// TwinCAT 3 PLC project Untitled1
// ProgramVersion: 3.1.4023.0
// libraries:
//   Tc2_Standard, * (Beckhoff Automation GmbH)
//   Tc2_System, * (Beckhoff Automation GmbH)
//   Tc3_Module, * (Beckhoff Automation GmbH)
// project tree:
//   Abstract Factory/ FB_AbstractFactory.TcPOU (not stored)
//   / Class Diagram.TcCD (not stored), PlcTask.TcTTO
//   Colors/ FB_Black.TcPOU (not stored), FB_Red.TcPOU (not stored), FB_Yellow.TcPOU (not stored)
//   Creator/ FB_ColorCreator.TcPOU (not stored), FB_ShapeCreator.TcPOU, FB_ShapeCreatorEX.TcPOU (not stored)
//   DUTs/ E_Color.TcDUT (not stored), E_Factory.TcDUT, E_Shape.TcDUT (not stored)
//   Factory Producer/ FB_FactoryProducer.TcPOU
//   Interfaces/ I_Color.TcIO, I_Shape.TcIO (not stored)
//   POUs/ MAIN.TcPOU
//   Shapes/ FB_Circle.TcPOU (not stored), FB_CustomShape.TcPOU (not stored), FB_Rectangle.TcPOU, FB_Square.TcPOU (not stored), FB_Star.TcPOU (not stored), FB_Triangle.TcPOU (not stored)
// real-time tasks:
//   TASK PlcTask: cycle T#10ms, priority 20, ADS port 350

CONFIGURATION Untitled1
    RESOURCE PLC ON TwinCAT3
        TASK PlcTask(INTERVAL := T#10ms, PRIORITY := 20);
        PROGRAM MAIN WITH PlcTask : MAIN;
    END_RESOURCE
END_CONFIGURATION

// ---- DUTs/E_Factory.TcDUT
{attribute 'qualified_only'}
{attribute 'strict'}
TYPE E_Factory :
(
	init := 0,
	Shape,
	Color,
	end
);
END_TYPE

// ---- Interfaces/I_Color.TcIO
INTERFACE I_Color

METHOD M_Fill : BOOL
VAR_INPUT
END_VAR
END_METHOD

END_INTERFACE

// ---- POUs/MAIN.TcPOU
PROGRAM MAIN
VAR
	fbFactoryProducer : FB_FactoryProducer;
	fbFactory : REFERENCE TO FB_AbstractFactory;
	
	iShape : I_Shape;
	iColor : I_Color;
	
	eShape : E_Shape := E_Shape.Star;
	eColor : E_Color := E_Color.Red;
	
	bStart1: BOOL;	
	bStart2: BOOL;	
END_VAR

IF bStart1 THEN
	//Draw
	fbFactory REF= fbFactoryProducer.M_GetFactory(eFactory := E_Factory.Shape);
	
	IF __ISVALIDREF(fbFactory) THEN
		iShape := fbFactory.M_GetShapeObject(eShape:=eShape);
	END_IF
	
	IF iShape <> 0 THEN
		iShape.M_Draw();
	END_IF
	
	//Fill
	fbFactory REF= fbFactoryProducer.M_GetFactory(eFactory := E_Factory.Color);
	
	IF __ISVALIDREF(fbFactory) THEN
		iColor := fbFactory.M_GetColorObject(eColor:=eColor);
	END_IF
	
	IF iColor <> 0 THEN
		iColor.M_Fill();
	END_IF
	
	//Release Memory
	fbFactoryProducer.M_ReleaseMemory();
	
	bStart1 := FALSE;
END_IF

//Alternatively, you can chain the methods and get the same result: 
IF bStart2 THEN
	fbFactoryProducer.M_GetFactory(eFactory := E_Factory.Shape).M_GetShapeObject(eShape:=eShape).M_Draw();
	fbFactoryProducer.M_GetFactory(eFactory := E_Factory.Color).M_GetColorObject(eColor:=eColor).M_Fill();
	
	//Release Memory
	fbFactoryProducer.M_ReleaseMemory();
	bStart2 := FALSE;
END_IF

END_PROGRAM

// ---- Factory Producer/FB_FactoryProducer.TcPOU
FUNCTION_BLOCK FB_FactoryProducer
VAR_INPUT
END_VAR
VAR_OUTPUT
END_VAR
VAR
	pColorFactoy : POINTER TO FB_ColorCreator;
	pShapeFactory : POINTER TO FB_ShapeCreator;
END_VAR

METHOD FB_exit : BOOL
VAR_INPUT
	bInCopyCode : BOOL; // if TRUE, the exit method is called for exiting an instance that is copied afterwards (online change).
END_VAR
IF pColorFactoy <> 0 THEN
	__DELETE(pColorFactoy);
	pColorFactoy := 0;
END_IF

IF pShapeFactory <> 0 THEN
	__DELETE(pShapeFactory);
	pShapeFactory := 0;
END_IF
END_METHOD

METHOD M_GetFactory : REFERENCE TO FB_AbstractFactory
VAR_INPUT
	eFactory : E_Factory;
END_VAR
CASE eFactory OF
	E_Factory.Color:
	
		pColorFactoy := __NEW(FB_ColorCreator);
		IF pColorFactoy <> 0 THEN
			M_GetFactory REF= (pColorFactoy^);
		END_IF
	
		eFactory := E_Factory.init;
	
	E_Factory.Shape:
	
		pShapeFactory := __NEW(FB_ShapeCreator);
		IF pShapeFactory <> 0 THEN
			M_GetFactory REF= (pShapeFactory^);
		END_IF

		eFactory := E_Factory.init;
	
END_CASE
END_METHOD

METHOD M_ReleaseMemory : BOOL
VAR_INPUT
END_VAR
IF pColorFactoy <> 0 THEN
	__DELETE(pColorFactoy);
	pColorFactoy := 0;
END_IF

IF pShapeFactory <> 0 THEN
	__DELETE(pShapeFactory);
	pShapeFactory := 0;
END_IF
END_METHOD

END_FUNCTION_BLOCK

// ---- Creator/FB_ShapeCreator.TcPOU
{attribute 'hide_all_locals'}
{attribute 'enable_dynamic_creation'}
FUNCTION_BLOCK FB_ShapeCreator  EXTENDS FB_AbstractFactory
VAR_INPUT
END_VAR
VAR_OUTPUT
END_VAR
VAR
      pCircle    : POINTER TO FB_Circle;
      pRectangle : POINTER TO FB_Rectangle;
      pSquare    : POINTER TO FB_Square;
      pStar      : POINTER TO FB_Star;
      pTriangle  : POINTER TO FB_Triangle;
      iShape 	 : I_Shape;
END_VAR

METHOD FB_exit : BOOL
VAR_INPUT
	bInCopyCode : BOOL; // if TRUE, the exit method is called for exiting an instance that is copied afterwards (online change).
END_VAR
IF (pCircle <> 0) THEN
  __DELETE(pCircle);
  pCircle := 0;
END_IF

IF (pRectangle <> 0) THEN
  __DELETE(pRectangle);
  pRectangle := 0;
END_IF

IF (pSquare <> 0) THEN
  __DELETE(pSquare);
  pSquare := 0;
END_IF

IF (pStar <> 0) THEN
  __DELETE(pStar);
  pStar := 0;
END_IF

IF (pTriangle <> 0) THEN
  __DELETE(pTriangle);
  pTriangle := 0;
END_IF
END_METHOD

METHOD M_GetShapeObject : I_shape
VAR_INPUT
	eShape : E_Shape;
END_VAR
CASE eShape OF
	E_Shape.Circle:
		
		//Dynamic instantiation  
		pCircle := __NEW(FB_Circle);
		iShape := pCircle^;
		
		//Return the object
		IF iShape <> 0 THEN
			M_GetShapeObject := iShape;
		END_IF
		
		//Release the memory
		IF (pCircle <> 0) THEN
			__DELETE(pCircle);
			pCircle := 0;
		END_IF
		
		eShape := E_Shape.init;
	
	E_Shape.Rectangle:
		pRectangle := __NEW(FB_Rectangle);
		iShape := pRectangle^;
		
		//Return the object
		IF iShape <> 0 THEN
			M_GetShapeObject := iShape;
		END_IF
		
		IF (pRectangle <> 0) THEN
			__DELETE(pRectangle);
			pRectangle := 0;
		END_IF
		
		eShape := E_Shape.init;	
		
	E_Shape.Sqaure:
		pSquare := __NEW(FB_Square);
		iShape := pSquare^;
		
		//Return the object
		IF iShape <> 0 THEN
			M_GetShapeObject := iShape;
		END_IF
		
		IF (pSquare <> 0) THEN
			__DELETE(pSquare);
			pSquare := 0;
		END_IF
		
		eShape := E_Shape.init;	

	E_Shape.Star:
		pStar := __NEW(FB_Star);
		iShape := pStar^;
		
		//Return the object
		IF iShape <> 0 THEN
			M_GetShapeObject := iShape;
		END_IF
		
		IF (pStar <> 0) THEN
			__DELETE(pStar);
			pStar := 0;
		END_IF
		
		eShape := E_Shape.init;	
	
	E_Shape.Triangle:
		pTriangle := __NEW(FB_Triangle);
		iShape := pTriangle^;
		
		//Return the object
		IF iShape <> 0 THEN
			M_GetShapeObject := iShape;
		END_IF
		
		IF (pTriangle <> 0) THEN
			__DELETE(pTriangle);
			pTriangle := 0;
		END_IF
		
		eShape := E_Shape.init;	
END_CASE
END_METHOD

METHOD M_ReleaseMemory : BOOL
VAR_INPUT
END_VAR
IF (pCircle <> 0) THEN
  __DELETE(pCircle);
  pCircle := 0;
END_IF

IF (pRectangle <> 0) THEN
  __DELETE(pRectangle);
  pRectangle := 0;
END_IF

IF (pSquare <> 0) THEN
  __DELETE(pSquare);
  pSquare := 0;
END_IF

IF (pStar <> 0) THEN
  __DELETE(pStar);
  pStar := 0;
END_IF

IF (pTriangle <> 0) THEN
  __DELETE(pTriangle);
  pTriangle := 0;
END_IF
END_METHOD

END_FUNCTION_BLOCK

// ---- Shapes/FB_Rectangle.TcPOU
{attribute 'enable_dynamic_creation'}
FUNCTION_BLOCK FB_Rectangle IMPLEMENTS I_Shape
VAR_INPUT
END_VAR
VAR_OUTPUT
END_VAR
VAR
END_VAR

{warning 'Agregar implementación de método'}
METHOD M_Draw : BOOL
ADSLOGSTR(ADSLOG_MSGTYPE_HINT, 'Draw rectangle', '');
M_Draw := TRUE;
END_METHOD

END_FUNCTION_BLOCK
